FUNCTION SetupHardware : BOOL
VAR
	iCardboardSlot : Cardboard;
	iCornerGuardSlot : CornerGuard;
	
	slotsArr : ARRAY[1..GVL.maxQueue] OF STRING;
	
	i : INT;
	j : INT;
END_VAR

FOR iCardboardSlot:=1 TO Cardboard.size-1 BY 1 DO
	slotsArr[iCardboardSlot] := TO_STRING(iCardboardSlot);
END_FOR
skidLeft.setupSlots(slotsArr);
skidRight.setupSlots(slotsArr);


FOR iCornerGuardSlot:=1 TO CornerGuard.size-1 BY 1 DO
	slotsArr[iCornerGuardSlot] := TO_STRING(iCornerGuardSlot);
END_FOR
magazineLeft.setupSlots(slotsArr);
magazineRight.setupSlots(slotsArr);

verticalDriveLeft.bEnable := 
verticalDriveRight.bEnable := 
horizontalDriveLeft.bEnable := 
horizontalDriveRight.bEnable := 
insertionBottom.bEnable := 
TRUE;

FOR i:=1 TO GVL.maxQueue BY 1 DO
	magazineLeft.setOccupancy(i := i, occupancy := IntegerBitAccess( TO_ULINT(robotLeft.inputs[3]), TO_ULINT(i-1)) );
	skidLeft.setOccupancy(i := i, occupancy := IntegerBitAccess( TO_ULINT(robotLeft.inputs[4]), TO_ULINT(i-1)) );
	
	magazineRight.setOccupancy(i := i, occupancy := IntegerBitAccess( TO_ULINT(robotRight.inputs[3]), TO_ULINT(i-1)) );
	skidRight.setOccupancy(i := i, occupancy := IntegerBitAccess( TO_ULINT(robotRight.inputs[4]), TO_ULINT(i-1)) );
END_FOR

END_FUNCTION

(* stored: Version 1.1.0.1, ProductVersion 3.1.4024.11
   POU SetupHardware: Id {ad70243f-26d6-4655-b24b-2a994d19bc18}, SpecialFunc None *)
